PROGRAM Faults
VAR
	faults_oneleft: ARRAY [1..5] OF WORD := [16#2A2A, 16#2A2A, 16#2A2A, 16#2A46, 16#4155];
	faults_oneRight: ARRAY [1..5] OF WORD := [16#4C54, 16#532A, 16#2A2A, 16#2A2A, 16#2A2A];
	
	door_1: ARRAY [1..5] OF WORD :=[16#446F, 16#6F72, 16#2031, 16#2020, 16#2020];
	door_2: ARRAY [1..5] OF WORD :=[16#446F, 16#6F72, 16#2032, 16#2020, 16#2020];
	door_3: ARRAY [1..5] OF WORD :=[16#446F, 16#6F72, 16#2033, 16#2020, 16#2020];
	door_4: ARRAY [1..5] OF WORD :=[16#446F, 16#6F72, 16#2034, 16#2020, 16#2020];
		
	
	
	pageNum: WORD := 0;	
END_VAR

(*IF GV_MODBUS.btnData = GV_MODBUS.btnUp THEN
	pageNum := pageNum - 1;
	
	IF pageNum < 0 THEN
		pageNum := 0;
	END_IF
	
	Execute_Write_Screen();
END_IF

IF GV_MODBUS.btnData = GV_MODBUS.btnDwn THEN
	pageNum := pageNum + 1;
	
	IF pageNum > 3 THEN
		pageNum := 3;
	END_IF
	
	Execute_Write_Screen();
END_IF

GV_MODBUS.oneLeft:= faults_oneLeft;
GV_MODBUS.oneRight:= faults_oneRight; 

IF pageNum = 0 THEN 
	                             
	GV_MODBUS.threeLeft:= up_limit; 
	
		GV_MODBUS.threeRight:= GV_MODBUS.fault_string;
	ELSE
		GV_MODBUS.threeRight:= GV_MODBUS.ok;		
	END_IF
	
	GV_MODBUS.twoLeft:= soft_up;
	
	IF GV_LIFT.CURRENT_POSITION < XML.savedvalues.UpSoftLim THEN
		GV_MODBUS.twoRight:= GV_MODBUS.fault_string;
	ELSE
		GV_MODBUS.twoRight:= GV_MODBUS.ok;	
		
	END_IF

	GV_MODBUS.fourLeft:= soft_down;
	IF GV_LIFT.CURRENT_POSITION < XML.savedvalues.DownSoftLim THEN
		GV_MODBUS.fourRight := GV_MODBUS.fault_string;
	ELSE
		GV_MODBUS.fourRight:= GV_MODBUS.ok;	
	END_IF
        
END_IF

IF pageNum = 1 THEN
	       	                        
	GV_MODBUS.twoLeft:= down_limit;
	IF GV_LIFT.DOWN_LIMIT_INDICATOR_OUT THEN
		GV_MODBUS.twoRight:= GV_MODBUS.fault_string;
	ELSE
		GV_MODBUS.twoRight:= GV_MODBUS.ok;
	END_IF	
            
	GV_MODBUS.threeLeft:= ult_limit;
	IF GV_LIFT.ULTIMATE_LIMIT_INDICATOR_OUT THEN
		GV_MODBUS.threeRight:= GV_MODBUS.fault_string;
	ELSE
		GV_MODBUS.threeRight:= GV_MODBUS.ok;
	END_IF     
                       
	GV_MODBUS.fourLeft:= door_1;
	IF GV_LIFT.DOOR_1_INDICATOR_OUT THEN
		GV_MODBUS.fourRight:= GV_MODBUS.fault_string;
	ELSE
		GV_MODBUS.fourRight:= GV_MODBUS.ok;
	END_IF  
   
END_IF

IF pageNum = 2 THEN
	                                
	GV_MODBUS.twoLeft:= door_2;
	IF GV_LIFT.DOOR_2_INDICATOR_OUT THEN
		GV_MODBUS.twoRight:= GV_MODBUS.fault_string;
	ELSE
		GV_MODBUS.threeRight:= GV_MODBUS.ok;
	END_IF	
                               
	GV_MODBUS.threeLeft:= door_3; 
	IF GV_LIFT.DOOR_3_INDICATOR_OUT THEN
		GV_MODBUS.threeRight:= GV_MODBUS.fault_string;
	ELSE
		GV_MODBUS.threeRight:= GV_MODBUS.ok;		
	END_IF
	               
	
	GV_MODBUS.fourLeft:= door_4;
	IF GV_LIFT.DOOR_4_INDICATOR_OUT THEN
		GV_MODBUS.fourRight:= GV_MODBUS.fault_string;
	ELSE
		GV_MODBUS.fourRight:= GV_MODBUS.ok;
	END_IF  
                           
	
END_IF

IF pageNum = 3 THEN
	GV_MODBUS.twoLeft := crush;
	
	IF GV_LIFT.CRUSH_PROTECTION_INDICATOR_OUT THEN
		GV_MODBUS.twoRight:= GV_MODBUS.fault_string;
	ELSE
		GV_MODBUS.twoRight:= GV_MODBUS.ok;
	END_IF	
	
	GV_MODBUS.threeLeft:= GV_MODBUS.blank;
	GV_MODBUS.threeRight:= GV_MODBUS.blank;
                               
	GV_MODBUS.fourLeft:= GV_MODBUS.blank; 
	GV_MODBUS.fourRight:= GV_MODBUS.blank;
	
END_IF


IF NOT GV_MODBUS.readExecute AND GV_MODBUS.addr = GV_MODBUS.oneLeftAddr THEN
	GV_MODBUS.data:= GV_MODBUS.oneLeft;
END_IF*)

END_PROGRAM

(* stored: Version 1.1.0.1, ProductVersion 3.1.4022.12
   POU Faults: Id {ff7267c4-369a-4e06-b636-9800277a52cd}, SpecialFunc None *)
